// TwinCAT 3 PLC project Untitled1
// ProgramVersion: 3.1.4023.0
// libraries:
//   Tc2_Standard, * (Beckhoff Automation GmbH)
//   Tc2_System, * (Beckhoff Automation GmbH)
//   Tc2_Utilities, * (Beckhoff Automation GmbH)
//   Tc3_Module, * (Beckhoff Automation GmbH)
// project tree:
//   GVLs/ GVL.TcGVL
//   / PlcTask.TcTTO
//   POUs/ MAIN.TcPOU
// real-time tasks:
//   TASK PlcTask: cycle T#10ms, priority 20, ADS port 350
//   TASK PlcTask1: cycle T#10ms, priority 21, ADS port 351

CONFIGURATION Untitled1
    RESOURCE PLC ON TwinCAT3
        TASK PlcTask(INTERVAL := T#10ms, PRIORITY := 20);
        PROGRAM MAIN WITH PlcTask : MAIN;
    END_RESOURCE
END_CONFIGURATION

// ---- GVLs/GVL.TcGVL
VAR_GLOBAL CONSTANT
	MAX_BUFFER_SIZE : UDINT := 1000;
END_VAR

// ---- POUs/MAIN.TcPOU
PROGRAM MAIN
VAR
	fbBufferOK : FB_MemRingBuffer;
	fbBufferReject : FB_MemRingBuffer;
	InData : LREAL;
	arrBuffer 	: ARRAY[0..MAX_BUFFER_SIZE] OF BYTE; (* Buffer memory used by FB_MemRingBuffer function block *)
	
	bOk			: BOOL;
	nCount		: UDINT;
	nLoad		: UDINT;
	outData			: LREAL;
	lastData: LREAL;
	bAdd: BOOL;
	bTest : BOOL;
END_VAR

IF bAdd THEN
	fbBufferOK.A_AddTail( pWrite:= ADR( InData ),
					cbWrite:= SIZEOF( InData ),
					pBuffer:= ADR( arrBuffer ),
					cbBuffer:= SIZEOF( arrBuffer ),
					bOk=> bOk,
					nCount => nCount );


	IF bOk THEN (* overflow ? *)
		bAdd := FALSE;
	END_IF
END_IF

fbBufferOK.A_GetHead( pRead:= ADR( outData ),
					cbRead:= SIZEOF( outData ),
					pBuffer:= ADR( arrBuffer ),
					cbBuffer:= SIZEOF( arrBuffer ),
					bOk=> bOk,
					nCount => nCount );
					
IF outData = 123 THEN
	bTest := TRUE;
	fbBufferOK.A_RemoveHead( 	pRead:= ADR( lastData ),
						cbRead:= SIZEOF( lastData ),
						pBuffer:= ADR( arrBuffer ),
						cbBuffer:= SIZEOF( arrBuffer ),
						bOk=> bOk,
						nCount => nCount );
END_IF

END_PROGRAM
